Staubli VAL3: clkValve0.pgx

program clkValve0()
begin
  call toggleValve(0)
end
